/// Axis move modulo parameter strucure
TYPE ST_AxisMoveModParameter EXTENDS ST_AxisMoveParameter :
STRUCT
	fPosition: LREAL;
	eDirection: MC_Direction;
END_STRUCT
END_TYPE

(* stored: Version 1.1.0.1, ProductVersion 3.1.4022.9
   DUT ST_AxisMoveModParameter: Id {dbd9f8cd-637c-467a-8153-f95b8d91b62c} *)
